(* PLC project SafeLOGIC, BrAutomation SafeDESIGNER  5.24.1.0 *)
(* stored: companyURL http://www.br-automation.com, creationDateTime Tue Oct 28 16:56:04 2025 *)

PROGRAM HeatWaterSys

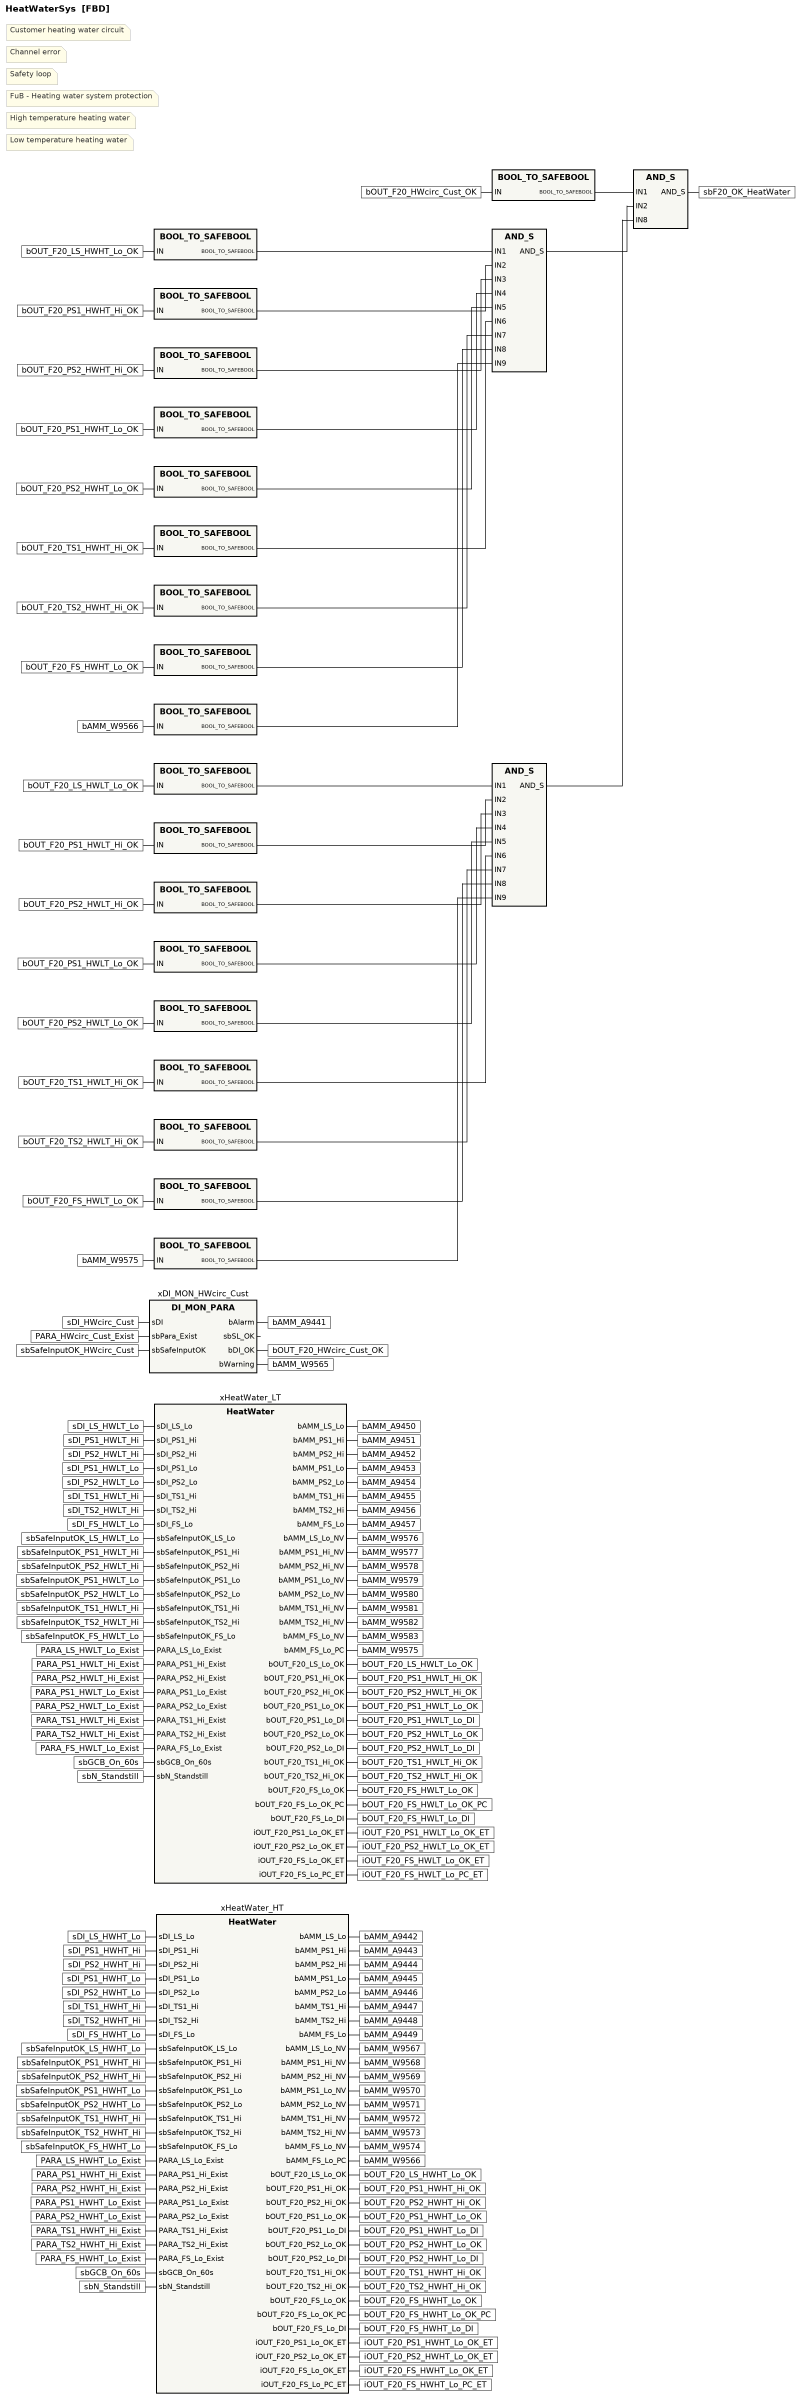
(* FBD diagram, written out as Structured Text *)
(* FuB - Heating water system protection *)
(* Customer heating water circuit *)
xDI_MON_HWcirc_Cust(sDI := sDI_HWcirc_Cust, sbPara_Exist := PARA_HWcirc_Cust_Exist, sbSafeInputOK := sbSafeInputOK_HWcirc_Cust);
bAMM_A9441 := xDI_MON_HWcirc_Cust.bAlarm;
(* Channel error *)
bAMM_W9565 := xDI_MON_HWcirc_Cust.bWarning;
bOUT_F20_HWcirc_Cust_OK := xDI_MON_HWcirc_Cust.bDI_OK;
(* High temperature heating water *)
xHeatWater_HT(sDI_LS_Lo := sDI_LS_HWHT_Lo, sDI_PS1_Hi := sDI_PS1_HWHT_Hi, sDI_PS2_Hi := sDI_PS2_HWHT_Hi, sDI_PS1_Lo := sDI_PS1_HWHT_Lo, sDI_PS2_Lo := sDI_PS2_HWHT_Lo, sDI_TS1_Hi := sDI_TS1_HWHT_Hi, sDI_TS2_Hi := sDI_TS2_HWHT_Hi, sDI_FS_Lo := sDI_FS_HWHT_Lo, sbSafeInputOK_LS_Lo := sbSafeInputOK_LS_HWHT_Lo, sbSafeInputOK_PS1_Hi := sbSafeInputOK_PS1_HWHT_Hi, sbSafeInputOK_PS2_Hi := sbSafeInputOK_PS2_HWHT_Hi, sbSafeInputOK_PS1_Lo := sbSafeInputOK_PS1_HWHT_Lo, sbSafeInputOK_PS2_Lo := sbSafeInputOK_PS2_HWHT_Lo, sbSafeInputOK_TS1_Hi := sbSafeInputOK_TS1_HWHT_Hi, sbSafeInputOK_TS2_Hi := sbSafeInputOK_TS2_HWHT_Hi, sbSafeInputOK_FS_Lo := sbSafeInputOK_FS_HWHT_Lo, PARA_LS_Lo_Exist := PARA_LS_HWHT_Lo_Exist, PARA_PS1_Hi_Exist := PARA_PS1_HWHT_Hi_Exist, PARA_PS2_Hi_Exist := PARA_PS2_HWHT_Hi_Exist, PARA_PS1_Lo_Exist := PARA_PS1_HWHT_Lo_Exist, PARA_PS2_Lo_Exist := PARA_PS2_HWHT_Lo_Exist, PARA_TS1_Hi_Exist := PARA_TS1_HWHT_Hi_Exist, PARA_TS2_Hi_Exist := PARA_TS2_HWHT_Hi_Exist, PARA_FS_Lo_Exist := PARA_FS_HWHT_Lo_Exist, sbGCB_On_60s := sbGCB_On_60s, sbN_Standstill := sbN_Standstill);
bAMM_A9442 := xHeatWater_HT.bAMM_LS_Lo;
bAMM_A9443 := xHeatWater_HT.bAMM_PS1_Hi;
bAMM_A9444 := xHeatWater_HT.bAMM_PS2_Hi;
bAMM_A9445 := xHeatWater_HT.bAMM_PS1_Lo;
bAMM_A9447 := xHeatWater_HT.bAMM_TS1_Hi;
bAMM_A9446 := xHeatWater_HT.bAMM_PS2_Lo;
bAMM_W9567 := xHeatWater_HT.bAMM_LS_Lo_NV;
bAMM_A9448 := xHeatWater_HT.bAMM_TS2_Hi;
bAMM_W9568 := xHeatWater_HT.bAMM_PS1_Hi_NV;
bAMM_A9449 := xHeatWater_HT.bAMM_FS_Lo;
bAMM_W9569 := xHeatWater_HT.bAMM_PS2_Hi_NV;
bAMM_W9570 := xHeatWater_HT.bAMM_PS1_Lo_NV;
bAMM_W9572 := xHeatWater_HT.bAMM_TS1_Hi_NV;
bAMM_W9573 := xHeatWater_HT.bAMM_TS2_Hi_NV;
bAMM_W9571 := xHeatWater_HT.bAMM_PS2_Lo_NV;
bAMM_W9574 := xHeatWater_HT.bAMM_FS_Lo_NV;
bOUT_F20_PS1_HWHT_Hi_OK := xHeatWater_HT.bOUT_F20_PS1_Hi_OK;
bAMM_W9566 := xHeatWater_HT.bAMM_FS_Lo_PC;
bOUT_F20_PS2_HWHT_Hi_OK := xHeatWater_HT.bOUT_F20_PS2_Hi_OK;
bOUT_F20_LS_HWHT_Lo_OK := xHeatWater_HT.bOUT_F20_LS_Lo_OK;
bOUT_F20_PS1_HWHT_Lo_OK := xHeatWater_HT.bOUT_F20_PS1_Lo_OK;
bOUT_F20_TS1_HWHT_Hi_OK := xHeatWater_HT.bOUT_F20_TS1_Hi_OK;
bOUT_F20_PS2_HWHT_Lo_OK := xHeatWater_HT.bOUT_F20_PS2_Lo_OK;
bOUT_F20_PS1_HWHT_Lo_DI := xHeatWater_HT.bOUT_F20_PS1_Lo_DI;
bOUT_F20_TS2_HWHT_Hi_OK := xHeatWater_HT.bOUT_F20_TS2_Hi_OK;
bOUT_F20_PS2_HWHT_Lo_DI := xHeatWater_HT.bOUT_F20_PS2_Lo_DI;
bOUT_F20_FS_HWHT_Lo_OK := xHeatWater_HT.bOUT_F20_FS_Lo_OK;
bOUT_F20_FS_HWHT_Lo_OK_PC := xHeatWater_HT.bOUT_F20_FS_Lo_OK_PC;
iOUT_F20_PS2_HWHT_Lo_OK_ET := xHeatWater_HT.iOUT_F20_PS2_Lo_OK_ET;
iOUT_F20_FS_HWHT_Lo_PC_ET := xHeatWater_HT.iOUT_F20_FS_Lo_PC_ET;
iOUT_F20_FS_HWHT_Lo_OK_ET := xHeatWater_HT.iOUT_F20_FS_Lo_OK_ET;
iOUT_F20_PS1_HWHT_Lo_OK_ET := xHeatWater_HT.iOUT_F20_PS1_Lo_OK_ET;
bOUT_F20_FS_HWHT_Lo_DI := xHeatWater_HT.bOUT_F20_FS_Lo_DI;
(* Low temperature heating water *)
xHeatWater_LT(sDI_LS_Lo := sDI_LS_HWLT_Lo, sDI_PS1_Hi := sDI_PS1_HWLT_Hi, sDI_PS2_Hi := sDI_PS2_HWLT_Hi, sDI_PS1_Lo := sDI_PS1_HWLT_Lo, sDI_PS2_Lo := sDI_PS2_HWLT_Lo, sDI_TS1_Hi := sDI_TS1_HWLT_Hi, sDI_TS2_Hi := sDI_TS2_HWLT_Hi, sDI_FS_Lo := sDI_FS_HWLT_Lo, sbSafeInputOK_LS_Lo := sbSafeInputOK_LS_HWLT_Lo, sbSafeInputOK_PS1_Hi := sbSafeInputOK_PS1_HWLT_Hi, sbSafeInputOK_PS2_Hi := sbSafeInputOK_PS2_HWLT_Hi, sbSafeInputOK_PS1_Lo := sbSafeInputOK_PS1_HWLT_Lo, sbSafeInputOK_PS2_Lo := sbSafeInputOK_PS2_HWLT_Lo, sbSafeInputOK_TS1_Hi := sbSafeInputOK_TS1_HWLT_Hi, sbSafeInputOK_TS2_Hi := sbSafeInputOK_TS2_HWLT_Hi, sbSafeInputOK_FS_Lo := sbSafeInputOK_FS_HWLT_Lo, PARA_LS_Lo_Exist := PARA_LS_HWLT_Lo_Exist, PARA_PS1_Hi_Exist := PARA_PS1_HWLT_Hi_Exist, PARA_PS2_Hi_Exist := PARA_PS2_HWLT_Hi_Exist, PARA_PS1_Lo_Exist := PARA_PS1_HWLT_Lo_Exist, PARA_PS2_Lo_Exist := PARA_PS2_HWLT_Lo_Exist, PARA_TS1_Hi_Exist := PARA_TS1_HWLT_Hi_Exist, PARA_TS2_Hi_Exist := PARA_TS2_HWLT_Hi_Exist, PARA_FS_Lo_Exist := PARA_FS_HWLT_Lo_Exist, sbGCB_On_60s := sbGCB_On_60s, sbN_Standstill := sbN_Standstill);
bAMM_A9450 := xHeatWater_LT.bAMM_LS_Lo;
bAMM_A9451 := xHeatWater_LT.bAMM_PS1_Hi;
bAMM_A9452 := xHeatWater_LT.bAMM_PS2_Hi;
bAMM_A9453 := xHeatWater_LT.bAMM_PS1_Lo;
bAMM_A9455 := xHeatWater_LT.bAMM_TS1_Hi;
bAMM_W9576 := xHeatWater_LT.bAMM_LS_Lo_NV;
bAMM_A9456 := xHeatWater_LT.bAMM_TS2_Hi;
bAMM_A9454 := xHeatWater_LT.bAMM_PS2_Lo;
bAMM_W9577 := xHeatWater_LT.bAMM_PS1_Hi_NV;
bAMM_A9457 := xHeatWater_LT.bAMM_FS_Lo;
bAMM_W9578 := xHeatWater_LT.bAMM_PS2_Hi_NV;
bAMM_W9579 := xHeatWater_LT.bAMM_PS1_Lo_NV;
bAMM_W9581 := xHeatWater_LT.bAMM_TS1_Hi_NV;
bAMM_W9582 := xHeatWater_LT.bAMM_TS2_Hi_NV;
bAMM_W9580 := xHeatWater_LT.bAMM_PS2_Lo_NV;
bOUT_F20_PS1_HWLT_Hi_OK := xHeatWater_LT.bOUT_F20_PS1_Hi_OK;
bOUT_F20_PS2_HWLT_Hi_OK := xHeatWater_LT.bOUT_F20_PS2_Hi_OK;
bOUT_F20_LS_HWLT_Lo_OK := xHeatWater_LT.bOUT_F20_LS_Lo_OK;
bAMM_W9583 := xHeatWater_LT.bAMM_FS_Lo_NV;
bAMM_W9575 := xHeatWater_LT.bAMM_FS_Lo_PC;
bOUT_F20_PS1_HWLT_Lo_OK := xHeatWater_LT.bOUT_F20_PS1_Lo_OK;
bOUT_F20_TS1_HWLT_Hi_OK := xHeatWater_LT.bOUT_F20_TS1_Hi_OK;
bOUT_F20_PS2_HWLT_Lo_OK := xHeatWater_LT.bOUT_F20_PS2_Lo_OK;
bOUT_F20_PS1_HWLT_Lo_DI := xHeatWater_LT.bOUT_F20_PS1_Lo_DI;
bOUT_F20_TS2_HWLT_Hi_OK := xHeatWater_LT.bOUT_F20_TS2_Hi_OK;
bOUT_F20_PS2_HWLT_Lo_DI := xHeatWater_LT.bOUT_F20_PS2_Lo_DI;
bOUT_F20_FS_HWLT_Lo_OK := xHeatWater_LT.bOUT_F20_FS_Lo_OK;
bOUT_F20_FS_HWLT_Lo_OK_PC := xHeatWater_LT.bOUT_F20_FS_Lo_OK_PC;
iOUT_F20_PS2_HWLT_Lo_OK_ET := xHeatWater_LT.iOUT_F20_PS2_Lo_OK_ET;
iOUT_F20_PS1_HWLT_Lo_OK_ET := xHeatWater_LT.iOUT_F20_PS1_Lo_OK_ET;
bOUT_F20_FS_HWLT_Lo_DI := xHeatWater_LT.bOUT_F20_FS_Lo_DI;
iOUT_F20_FS_HWLT_Lo_PC_ET := xHeatWater_LT.iOUT_F20_FS_Lo_PC_ET;
iOUT_F20_FS_HWLT_Lo_OK_ET := xHeatWater_LT.iOUT_F20_FS_Lo_OK_ET;
(* Safety loop *)
sbF20_OK_HeatWater := AND_S(BOOL_TO_SAFEBOOL(bOUT_F20_HWcirc_Cust_OK), AND_S(BOOL_TO_SAFEBOOL(bOUT_F20_LS_HWHT_Lo_OK), BOOL_TO_SAFEBOOL(bOUT_F20_PS1_HWHT_Hi_OK), BOOL_TO_SAFEBOOL(bOUT_F20_PS2_HWHT_Hi_OK), BOOL_TO_SAFEBOOL(bOUT_F20_PS1_HWHT_Lo_OK), BOOL_TO_SAFEBOOL(bOUT_F20_PS2_HWHT_Lo_OK), BOOL_TO_SAFEBOOL(bOUT_F20_TS1_HWHT_Hi_OK), BOOL_TO_SAFEBOOL(bOUT_F20_TS2_HWHT_Hi_OK), BOOL_TO_SAFEBOOL(bOUT_F20_FS_HWHT_Lo_OK), BOOL_TO_SAFEBOOL(bAMM_W9566)), AND_S(BOOL_TO_SAFEBOOL(bOUT_F20_LS_HWLT_Lo_OK), BOOL_TO_SAFEBOOL(bOUT_F20_PS1_HWLT_Hi_OK), BOOL_TO_SAFEBOOL(bOUT_F20_PS2_HWLT_Hi_OK), BOOL_TO_SAFEBOOL(bOUT_F20_PS1_HWLT_Lo_OK), BOOL_TO_SAFEBOOL(bOUT_F20_PS2_HWLT_Lo_OK), BOOL_TO_SAFEBOOL(bOUT_F20_TS1_HWLT_Hi_OK), BOOL_TO_SAFEBOOL(bOUT_F20_TS2_HWLT_Hi_OK), BOOL_TO_SAFEBOOL(bOUT_F20_FS_HWLT_Lo_OK), BOOL_TO_SAFEBOOL(bAMM_W9575)));
END_PROGRAM
